// TIA Portal V20 export
DATA_BLOCK "DB_CC_Main"   // DB101
// stored: AutoNumber false, InstanceOfName CC_Main, InstanceOfType FB
"CC_Main"
   // VAR_INPUT
   //    HMI_Reset : Bool;
   //    ST23_Selected : Bool;
   //    CNT_DownPos1 : Bool;
   //    CNT_DownPos2 : Bool;
   //    CNT_UpPos1 : Bool;
   //    CNT_UpPos2 : Bool;
   //    Hydraulic_Roller_DownPos1 : Bool;
   //    Hydraulic_Roller_DownPos2 : Bool;
   //    Hydraulic_Roller_UpPos1 : Bool;
   //    Hydraulic_Roller_UpPos2 : Bool;
   //    Drive_Roller_DownPos1 : Bool;
   //    Drive_Roller_DownPos2 : Bool;
   //    Drive_Roller_UpPos1 : Bool;
   //    Drive_Roller_UpPos2 : Bool;
   //    Module_DownPos1 : Bool;
   //    Module_DownPos2 : Bool;
   //    Module_UpPos1 : Bool;
   //    Module_UpPos2 : Bool;
   // END_VAR
   // VAR_OUTPUT
   //    Hydraulic_Main_Valve_Control : Bool;
   // END_VAR
   // VAR
   //    Hydraulic_Unit_Active : Bool;
   //    Any_Valve_Active : Bool;
   //    HydUnitTimerOff { S7_SetPoint := 'True'} : TON_TIME;
   //    HydraulicUnit_MC_Power { S7_SetPoint := 'True'} : MC_POWER;
   //    HydraulicUnit_MC_MoveJog { S7_SetPoint := 'True'} : MC_MOVEJOG;
   //    HydraulicUnit_MC_Reset { S7_SetPoint := 'True'} : MC_RESET;
   //    Vibrator_Control_MOD1 { S7_SetPoint := 'True'} : "CC_Vibrator_Control";
   //    Vibrator_Control_MOD2 { S7_SetPoint := 'True'} : "CC_Vibrator_Control";
   //    Vibrator_Control_MOD3 { S7_SetPoint := 'True'} : "CC_Vibrator_Control";
   //    Module_Control_ST23 { S7_SetPoint := 'True'} : "CC_Vib_Modules";
   //    ST23_UP_whenMoving { S7_SetPoint := 'True'} : Bool;
   //    ST24_UP_whenMoving : Bool;
   //    ST25_UP_whenMoving : Bool;
   //    MC_Power_Vib1 { S7_SetPoint := 'True'} : MC_POWER;
   //    MC_RESET_Vib1 { S7_SetPoint := 'True'} : MC_RESET;
   //    MC_MOVEJOG_Vib1 { S7_SetPoint := 'True'} : MC_MOVEJOG;
   //    ST24_DriveRollsUP { S7_SetPoint := 'True'} : Bool;
   //    ST24_DriveRollsDown : Bool;
   //    ST25_DriveRollsUp : Bool;
   //    ST25_DriveRollsDown : Bool;
   //    ST23_Station_Control { S7_SetPoint := 'True'} : "CC_Station_Control";
   //    ST24_Station_Control { S7_SetPoint := 'True'} : "CC_Station_Control";
   //    ST25_Station_Control { S7_SetPoint := 'True'} : "CC_Station_Control";
   //    ST24_Selected : Bool;
   // END_VAR
BEGIN
END_DATA_BLOCK
